// TIA Portal V17 export
FUNCTION "串联_触点线圈" : Void   // FC, LAD
{ S7_Optimized_Access := 'TRUE' }
VERSION : 0.1
// stored: AutoNumber true, IsIECCheckEnabled false, SetENOAutomatically false
BEGIN

REGION Network 1
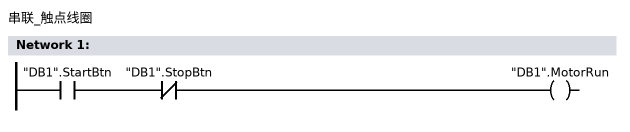
   RUNG wire#powerrail
      Contact( "DB1".StartBtn )
      I_Contact( "DB1".StopBtn )
      Coil( "DB1".MotorRun )
   END_RUNG
   // the same network as SCL:
   "DB1".MotorRun := "DB1".StartBtn AND NOT "DB1".StopBtn;
END_REGION
END_FUNCTION
